INTERFACE I_PersistentEventStorage

METHOD StoreEvent
VAR_INPUT
	stEvent : ST_Event;
END_VAR
END_METHOD

END_INTERFACE

(* stored: Version 1.1.0.1, ProductVersion 3.1.4024.12
   Itf I_PersistentEventStorage: Id {5c88885c-75be-4a05-9856-e14ff134a965}
   Method StoreEvent: Id {fc0850ef-9427-4bb8-90dd-f3aca46b7050} *)
